# EPICS autosave request: dxpApp/Db/dxpMapping_settings.req
$(P)CollectMode
$(P)ListMode
$(P)PixelAdvanceMode
$(P)PixelsPerRun
$(P)AutoPixelsPerBuffer
$(P)PixelsPerBuffer
$(P)IgnoreGate
$(P)SyncCount
$(P)InputLogicPolarity
$(P)SyncMasterChannel
$(P)GateMasterChannel
$(P)LBUSMasterChannel
